(* CoDeSys 2.3.9.62 project: main.pro *)
(* Libraries: Standard.lib, Iecsfc.lib 8.11.10 11:37:48, SYSLIBCALLBACK.LIB *)

(* PLC configuration (modules and I/O channels)
K-Bus [K_Bus] node 0, in %IB0 out %QB0
input1 AT %IX0.0 [BOOLOnX_I] Ch_1 Digital input
input2 AT %IX0.1 [BOOLOnX_I] Ch_2 Digital input
input3 AT %IX0.2 [BOOLOnX_I] Ch_3 Digital input
input4 AT %IX0.3 [BOOLOnX_I] Ch_4 Digital input
input5 AT %IX0.4 [BOOLOnX_I] Ch_5 Digital input
input6 AT %IX0.5 [BOOLOnX_I] Ch_6 Digital input
input7 AT %IX0.6 [BOOLOnX_I] Ch_7 Digital input
input8 AT %IX0.7 [BOOLOnX_I] Ch_8 Digital input
outPut1 AT %QX0.0 [BOOLOnX_Q] Ch_1 Digital output
outPut2 AT %QX0.1 [BOOLOnX_Q] Ch_2 Digital output
AT %QX0.2 [BOOLOnX_Q] Ch_3 Digital output
AT %QX0.3 [BOOLOnX_Q] Ch_4 Digital output
AT %QX0.4 [BOOLOnX_Q] Ch_5 Digital output
AT %QX0.5 [BOOLOnX_Q] Ch_6 Digital output
AT %QX0.6 [BOOLOnX_Q] Ch_7 Digital output
AT %QX0.7 [BOOLOnX_Q] Ch_8 Digital output
Internal Digital I/O [InternalDigIO] node 1, in %IB512 out %QB512
  Internal Digital Inputs [Internal_DIN] node 0, in %IB512 out %QB512
    DIN1 AT %IX2300.0 [BOOLOnX_I] Internal Digital Input Bit 1
    DIN2 AT %IX2300.1 [BOOLOnX_I] Internal Digital Input Bit 2
  Internal Digital Outputs [Internal_DOUT] node 1, in %IB513 out %QB512
    DOUT1 AT %QX2300.0 [BOOLOnX_Q] Internal Digital Output Bit 1
    DOUT2 AT %QX2300.1 [BOOLOnX_Q] Internal Digital Output Bit 2
Fieldbus variables [FB_VARS] node 3, in %IB0 out %QB0
Flag variables [FLAG_VARS] node 4, in %IB0 out %QB0
Modbus-Master [MB_MASTER] node 5, in %IB0 out %QB0
*)

(* Task configuration *)
TASK main (PRIORITY := 15, INTERVAL := T#50ms);
	main();
END_TASK

(* POU main, ST *)
PROGRAM main
VAR

	inv0 : BOOL;
	inv1 : BOOL;
	inv2 : BOOL;
	inv3: BOOL;
	inv4: BOOL;
	inv5: BOOL;
	inv6: BOOL;
	inv7: BOOL;

	outputByte : BYTE;


	roll : LREAL := 1;
	pitch : LREAL := 2;

	angle0 : LREAL;
	angle1 : LREAL;
	angle2 : LREAL;

	didBound : BOOL;

	angleFunction : ComputeMotorAngles;

END_VAR
outPut1 := TRUE;

inv0 := input1;
inv1 := input2;
inv2 := input3;
inv3 := input4;
inv4 := input5;
inv5 := input6;
inv6 := input7;
inv7 := input8;

outputByte := Byte9;

angleFunction.roll := roll;
angleFunction.pitch := pitch;

angleFunction();

angle0 := angleFunction.angle0;
angle1 := angleFunction.angle1;
angle2 := angleFunction.angle2;
didBound := angleFunction.didBound;
END_PROGRAM

(* POU ComputeMotorAngles, ST *)
FUNCTION_BLOCK ComputeMotorAngles
VAR_INPUT
	roll : LREAL;
	pitch : LREAL;
END_VAR
VAR_OUTPUT
	angle0 : LREAL;
	angle1 : LREAL;
	angle2 : LREAL;

	didBound : BOOL;
END_VAR
VAR
	l : LREAL := 1.75;
	delta : LREAL := 0.08;
	s0 : LREAL := 1.0;
	s1 : LREAL := 1.0;

	tmpVar : LREAL;

	p0 : LREAL;
	p1 : LREAL;
	p2 : LREAL;
END_VAR
tmpVar := l / 2 * ATAN(pitch / s1);
p1 :=delta + tmpVar;
p0 := delta - tmpVar;

p2 := delta - (l * SQRT(3) / 2) * ATAN(roll / s0);

p0 := -1.0 * (p0 - delta) / delta;
p1 := -1.0 * (p1 - delta) / delta;
p2 := -1.0 * (p2 - delta) / delta;

didBound := FALSE;

IF (p0 > 1.0) THEN
	p0 := 1.0;
	didBound := TRUE;
ELSIF (p0 < -1.0) THEN
	p0 := -1.0;
	didBound := TRUE;
END_IF


IF (p1 > 1.0) THEN
	p1 := 1.0;
	didBound := TRUE;
ELSIF (p1 < -1.0) THEN
	p1 := -1.0;
	didBound := TRUE;
END_IF

IF (p2 > 1.0) THEN
	p2 := 1.0;
	didBound := TRUE;
ELSIF (p2 < -1.0) THEN
	p2 := -1.0;
	didBound := TRUE;
END_IF

angle0 := ACOS(p0);
angle1 := ACOS(p1);
angle2 := ACOS(p2);
END_FUNCTION_BLOCK

(* POU Configuration/MODBUS_CONFIGURATION, ST *)
PROGRAM MODBUS_CONFIGURATION        
VAR                                
END_VAR                            
(*                                 
   <?xml version="1.0" encoding="UTF-16" standalone="yes"?>
<network xml_structure_version="1" xml_feature_version="1">
	<generator_settings minRTUTaskCycleTimeMs="5" minEthaskCycleTimeMs="5" ethSlaveMultiplier="0.1" rtuInterfaceMultiplier="0.1" taskGeneration="true"/>
</network>
                              
*)                                 
;                                  
END_PROGRAM
